(* PLC project Unnamed, Unknown Unnamed 1 *)
(* stored: creationDateTime 2026-05-25T17:31:08, modificationDateTime 2026-05-25T17:31:08 *)

PROGRAM main
  VAR
    MainGreen : BOOL := True;
    MainYellow : BOOL := False;
    MainRed : BOOL := False;
    SideGreen : BOOL := False;
    SideYellow : BOOL := False;
    SideRed : BOOL := True;
    CarWaiting : BOOL := False;
    PedWaiting : BOOL := False;
    GreenTimer : TON;
    YellowTimer : TON;
    SideGreenTimer : TON;
    SideYellowTimer : TON;
  END_VAR

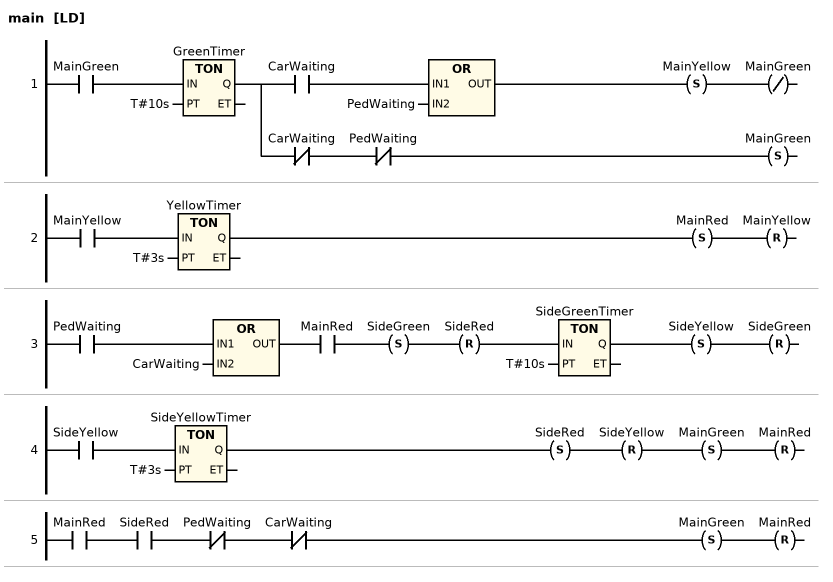
(* LD diagram, written out as Structured Text *)
GreenTimer(IN := MainGreen, PT := T#10s);
IF GreenTimer.Q AND CarWaiting OR PedWaiting THEN MainYellow := TRUE; END_IF;
MainGreen := NOT (GreenTimer.Q AND CarWaiting OR PedWaiting);
IF GreenTimer.Q AND NOT CarWaiting AND NOT PedWaiting THEN MainGreen := TRUE; END_IF;
YellowTimer(IN := MainYellow, PT := T#3s);
IF YellowTimer.Q THEN MainRed := TRUE; END_IF;
IF YellowTimer.Q THEN MainYellow := FALSE; END_IF;
IF MainRed AND SideRed AND NOT PedWaiting AND NOT CarWaiting THEN MainGreen := TRUE; END_IF;
IF MainRed AND SideRed AND NOT PedWaiting AND NOT CarWaiting THEN MainRed := FALSE; END_IF;
IF (PedWaiting OR CarWaiting) AND MainRed THEN SideGreen := TRUE; END_IF;
IF (PedWaiting OR CarWaiting) AND MainRed THEN SideRed := FALSE; END_IF;
SideGreenTimer(IN := (PedWaiting OR CarWaiting) AND MainRed, PT := T#10s);
IF SideGreenTimer.Q THEN SideYellow := TRUE; END_IF;
IF SideGreenTimer.Q THEN SideGreen := FALSE; END_IF;
SideYellowTimer(IN := SideYellow, PT := T#3s);
IF SideYellowTimer.Q THEN SideRed := TRUE; END_IF;
IF SideYellowTimer.Q THEN SideYellow := FALSE; END_IF;
IF SideYellowTimer.Q THEN MainGreen := TRUE; END_IF;
IF SideYellowTimer.Q THEN MainRed := FALSE; END_IF;
END_PROGRAM

CONFIGURATION Config0
  RESOURCE Res0 ON PLC
    TASK task0(INTERVAL := T#20ms, PRIORITY := 1);
    PROGRAM instance0 WITH task0 : main;
  END_RESOURCE
END_CONFIGURATION
